FUNCTION F_ResetExternalFunctionError : BOOL
(**************************************************************************************
 * 	Application		:	BoxControl Framework
 *	Revision		:	$Revision: 404529 $
 *	Revision date	:	$Date: 2018-04-23 08:21:38 +0200 (Mo., 23 Apr 2018) $
 *	Last changed by	:	$Author: b7bolm $
 *	URL				:	$URL: http://almscdc.swisslog.com/repo/SWPD/Development/BoxControlFramework/20_Release/trunk/01_Software/BCF/BCF/JumpStart/20_Product/10_App/12_E_Functions/10_Lib/10_Conv/10_Functions/F_ResetExternalFunctionError.TcPOU $
 *
 *	Purpose			:	Reset external error
 *						Add an External error, which will be reported over the configured
 *						position.
 *						
 *
 * ------------------------------------------------------------------------------------
 *	Copyright Swisslog [IP AG], Switzerland. All rights reserved.
 * 
 * ------------------------------------------------------------------------------------
 *	
 * 	Revision History: 
 *
 * 	VERSION			DATE			INITIALS			DESCRIPTION
 *	0.1				01.01.2001		swl					Example
 *
 **************************************************************************************)
VAR_INPUT
	eFunctionNumber : E_FunctionNumber; 
	ZoneNumber		: INT;
	Reset			: BOOL;
END_VAR


// Validate inputs
IF eFunctionNumber > E_FunctionNumber.F_BEGIN_FUNCTION THEN
	IF __ISVALIDREF(FunctionRegistry[eFunctionNumber].rFunction) THEN
		// Reset external error on instance
		FunctionRegistry[eFunctionNumber].rFunction.M_ResetExternalError(
			mZoneNumber := ZoneNumber,
			mReset := Reset);
	END_IF
END_IF

END_FUNCTION

(* stored: Version 1.1.0.1, ProductVersion 3.1.4022.12
   POU F_ResetExternalFunctionError: Id {cb22b2d8-5ff5-4030-bf62-3ea558d10caf}, SpecialFunc None *)
